{attribute addProperty BoxType "KL2641"}
{attribute addProperty Id "Channel_1Channel_047EC78B00"}
{attribute addProperty CRC "2898456704"}
{attribute addProperty SizeInBites "0"}
{attribute addProperty SizeInBytes "0"}
TYPE KL2641_ACC2F080 :
STRUCT
	{attribute addProperty Name "Channel_1"}
	Channel_1 : Channel_047EC78B;
END_STRUCT
END_TYPE

(* stored: Version 1.2.0.0, ProductVersion 3.1.4024.9
   DUT KL2641_ACC2F080: Id {09ab859b-3ac3-4a6c-a62c-c4b505d7fa63} *)
